PROGRAM prgComLynus
VAR
	fbCom			: FB_MqttCommunicator;
END_VAR

fbCom(
	bConnect:= TRUE, 
	sUserName:= 'b70e88c8-0481-4d36-92fe-45daf83d392d', 
	sUserPassword:= '31c9e512-5d63-471e-8e0c-6ecec0b71d43', 
	eSavePositionCertificate:= eSavePositionOnPLC.ePostionHardDisk, 
	bConnected=> , 
	bError=> , 
	hrErrorCode=> , 
	eConnectionState=> , 
	eErrorMessage_Out=> );

END_PROGRAM

(* stored: Version 1.1.0.1, ProductVersion 3.1.4024.9
   POU prgComLynus: Id {63d49923-762f-40e3-a7f4-737e68cbccfe}, SpecialFunc None *)
